TYPE csp_case_feed_magazine_level_enum :(
	CSP_CASE_FEED_MAGAZINE_LEVEL_STATUS_IDLE						:= 0,
	CSP_CASE_FEED_MAGAZINE_LEVEL_STATUS_ZONE4						:= 1,
	CSP_CASE_FEED_MAGAZINE_LEVEL_STATUS_ZONE3						:= 2,
	CSP_CASE_FEED_MAGAZINE_LEVEL_STATUS_ZONE2						:= 3,
	CSP_CASE_FEED_MAGAZINE_LEVEL_STATUS_ZONE1						:= 4,
	CSP_CASE_FEED_MAGAZINE_LEVEL_STATUS_LOW							:= 5,
	CSP_CASE_FEED_MAGAZINE_LEVEL_STATUS_MIN							:= 6,
	CSP_CASE_FEED_MAGAZINE_LEVEL_STATUS_UNDER_MIN					:= 7
    ) := CSP_CASE_FEED_MAGAZINE_LEVEL_STATUS_IDLE;
END_TYPE

(* stored: Version 1.1.0.1, ProductVersion 3.1.4024.3
   DUT csp_case_feed_magazine_level_enum: Id {23a10748-dbbb-4505-b78c-5c7513aca255} *)
